// TIA Portal V20 export
DATA_BLOCK "SBK10"   // DB328
// stored: MemoryReserve 100
   VAR
      "SAFETY DOOR LOCK7.INPUT" : Bool := TRUE;
      "SAFETY DOOR LOCK8.INPUT" : Bool := TRUE;
      SPARE : Bool := TRUE;
      SPARE_1 : Bool := FALSE;
      "SAFETY DOOR LOCK7.INPUT_1" : Bool := FALSE;
      "SAFETY DOOR LOCK8.INPUT_1" : Bool := FALSE;
      SPARE_2 : Bool := FALSE;
      SPARE_3 : Bool := FALSE;
      "SAFETY DOOR LOCK7.OUTPUT" : Bool := FALSE;
      "SAFETY DOOR LOCK8.OUTPUT" : Bool := FALSE;
      SPARE_4 : Bool := FALSE;
   END_VAR
BEGIN
END_DATA_BLOCK
